INTERFACE I_Analog

PROPERTY AnalogSignal : INT
GET
END_GET
SET
END_SET
END_PROPERTY

METHOD Scale : BOOL
VAR_INPUT
END_VAR
END_METHOD

PROPERTY ScaledAnalog : INT
GET
END_GET
SET
END_SET
END_PROPERTY

END_INTERFACE

(* stored: Version 1.1.0.1, ProductVersion 3.1.4024.12
   Itf I_Analog: Id {e5efea24-2bcb-4cf4-b329-1255d100a501}
   Property AnalogSignal: Id {c0b94fb5-afa8-4ee2-a0b0-a233a53f3251}
   Get Get: Id {aa692638-df91-42ce-8188-59ed7b6a96e4}
   Set Set: Id {3742b2fd-22f3-4535-b280-1463e96d076c}
   Method Scale: Id {aad8d38f-fb15-45fb-b2e7-72a4db2df1fc}
   Property ScaledAnalog: Id {b1d8e986-1d3b-4e52-b121-13b18448f590}
   Get Get: Id {f8d648b0-df73-4cca-9e7e-143d0f6ed8e8}
   Set Set: Id {ee9f6acd-689c-4f45-9373-352444588549} *)
